{attribute 'GeneratedUsingTerminal: EL2564-0000-0016'}
{attribute addProperty BoxType "EL2564-0000-0016"}
{attribute addProperty Id "WarningBOOL1ErrorBOOL1TxPDO_ToggleBOOL1"}
{attribute addProperty CRC "1809415223"}
{attribute addProperty Size "3"}
TYPE Status_6BD97C37 :
STRUCT
	{attribute addProperty Name "Warning"}
	Warning : BOOL;
	{attribute addProperty Name "Error"}
	Error : BOOL;
	{attribute addProperty Name "TxPDO_Toggle"}
	TxPDO_Toggle : BOOL;
END_STRUCT
END_TYPE

(* stored: Version 1.2.0.0, ProductVersion 3.1.4024.9
   DUT Status_6BD97C37: Id {f77fea23-faf7-4fc4-a679-0d174d783ed4} *)
